SYSTEM QUERY_TEST (* Test QUERY Function in Remote Devices *)
  (* Standard: 61499 ITA; Function: QUERY Functional Test *)
  (* Version 0.0, 2001-11-24, JHC, Rockwell Automation *)
  APPLICATION TEST
    FBS
      SELECT : IN_CHOICE;
      GEN : QUERY_GEN;
      QTEXT : IN_TEXT_S;
      QUERY : IN_EVENT;
      CLIENT : CLIENT_2_1;
      RTEXT : OUT_TEXT_S;
    END_FBS
    EVENT_CONNECTIONS
      SELECT.INITO TO QUERY.INIT;
      QUERY.INITO TO GEN.REQ;
      GEN.CNF TO QTEXT.INIT;
      QTEXT.INITO TO CLIENT.INIT;
      CLIENT.INITO TO RTEXT.INIT;
      SELECT.IND TO GEN.REQ;
      QTEXT.CNF TO CLIENT.REQ;
      CLIENT.CNF TO RTEXT.REQ;
    END_CONNECTIONS
    DATA_CONNECTIONS
      "FB,Connection" TO SELECT.CHOICES;
      SELECT.I TO GEN.N;
      QTEXT.OUT TO CLIENT.SD_2;
      CLIENT.RD_1 TO RTEXT.IN;
      1 TO SELECT.QI;
      1 TO QTEXT.QI;
      1 TO QUERY.QI;
      1 TO CLIENT.QI;
      1 TO RTEXT.QI;
      "QUERY" TO QUERY.LABEL;
      "localhost:61494" TO CLIENT.ID;
      "RUT" TO GEN.DSTI;
      GEN.DSTO TO CLIENT.SD_1;
      GEN.QUERY TO QTEXT.IVAL;
    END_CONNECTIONS
  END_APPLICATION
  DEVICE QUERY_TESTER : FRAME_DEVICE
    RESOURCE RES1 : PANEL_RESOURCE
      FBS
        SELECT : IN_CHOICE;
        QUERY : IN_EVENT;
        GEN : QUERY_GEN;
        QTEXT : IN_TEXT_S;
        CLIENT : CLIENT_2_1;
        RTEXT : OUT_TEXT_S;
      END_FBS
      EVENT_CONNECTIONS
        START.COLD TO SELECT.INIT;
        START.WARM TO SELECT.INIT;
        SELECT.INITO TO QUERY.INIT;
        QUERY.INITO TO GEN.REQ;
        SELECT.IND TO GEN.REQ;
        GEN.CNF TO QTEXT.INIT;
        QTEXT.INITO TO CLIENT.INIT;
        QUERY.IND TO QTEXT.REQ;
        QTEXT.CNF TO CLIENT.REQ;
        CLIENT.INITO TO RTEXT.INIT;
        CLIENT.CNF TO RTEXT.REQ;
      END_CONNECTIONS
      DATA_CONNECTIONS
        "FB,Connection" TO SELECT.CHOICES;
        1 TO SELECT.QI;
        1 TO QUERY.QI;
        "QUERY" TO QUERY.LABEL;
        SELECT.I TO GEN.N;
        1 TO QTEXT.QI;
        QTEXT.OUT TO CLIENT.SD_2;
        1 TO CLIENT.QI;
        "localhost:61494" TO CLIENT.ID;
        "RUT" TO GEN.DSTI;
        GEN.DSTO TO CLIENT.SD_1;
        CLIENT.RD_1 TO RTEXT.IN;
        1 TO RTEXT.QI;
        [4,40] TO QTEXT.SIZE;
        GEN.QUERY TO QTEXT.IVAL;
        [6,40] TO RTEXT.SIZE;
      END_CONNECTIONS
    END_RESOURCE
    DATA_CONNECTIONS
      1 TO RES1.TRACE;
    END_CONNECTIONS
  END_DEVICE
  DEVICE DUT : RMT_FRAME (* Device Under Test *)
    RESOURCE RUT : PANEL_RESOURCE (* Resource Under Test *)
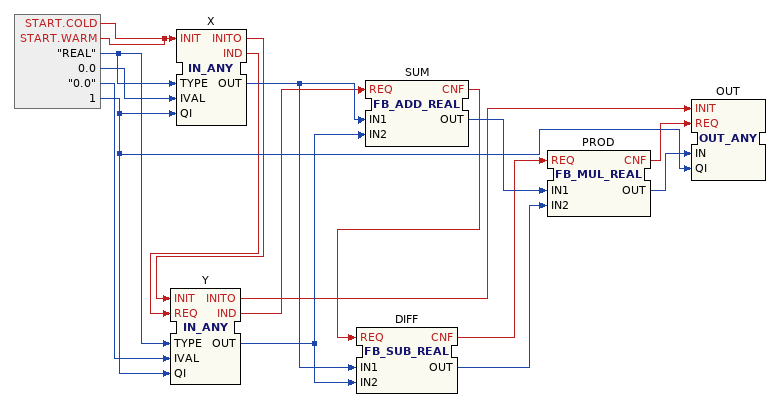
      FBS
        X : IN_ANY;
        Y : IN_ANY;
        SUM : FB_ADD_REAL;
        DIFF : FB_SUB_REAL;
        PROD : FB_MUL_REAL;
        OUT : OUT_ANY; (* X**2-Y**2 *)
      END_FBS
      EVENT_CONNECTIONS
        START.COLD TO X.INIT;
        START.WARM TO X.INIT;
        X.INITO TO Y.INIT;
        Y.INITO TO OUT.INIT;
        X.IND TO Y.REQ;
        Y.IND TO SUM.REQ;
        SUM.CNF TO DIFF.REQ;
        DIFF.CNF TO PROD.REQ;
        PROD.CNF TO OUT.REQ;
      END_CONNECTIONS
      DATA_CONNECTIONS
        X.OUT TO SUM.IN1;
        X.OUT TO DIFF.IN1;
        Y.OUT TO SUM.IN2;
        Y.OUT TO DIFF.IN2;
        SUM.OUT TO PROD.IN1;
        DIFF.OUT TO PROD.IN2;
        PROD.OUT TO OUT.IN;
        "REAL" TO X.TYPE;
        0.0 TO X.IVAL;
        "REAL" TO Y.TYPE;
        "0.0" TO Y.IVAL;
        1 TO X.QI;
        1 TO Y.QI;
        1 TO OUT.QI;
      END_CONNECTIONS
    END_RESOURCE
  END_DEVICE
  DATA_CONNECTIONS (* parameter values *)
    [375,50,100,150] TO DUT.BOUNDS;
    [1,1] TO DUT.GRID;
    "localhost:61494" TO DUT.MGR_ID;
    [50,50,325,240] TO QUERY_TESTER.BOUNDS;
    [1,1] TO QUERY_TESTER.GRID;
  END_CONNECTIONS
  MAPPINGS
    TEST.SELECT ON QUERY_TESTER.RES1.SELECT;
    TEST.QUERY ON QUERY_TESTER.RES1.QUERY;
    TEST.GEN ON QUERY_TESTER.RES1.GEN;
    TEST.QTEXT ON QUERY_TESTER.RES1.QTEXT;
    TEST.CLIENT ON QUERY_TESTER.RES1.CLIENT;
    TEST.RTEXT ON QUERY_TESTER.RES1.RTEXT;
  END_MAPPINGS
END_SYSTEM
